Fanuc KAREL source: kb00158.KL

-- PROVISIONAL review KL for V770-1; original PC SHA256 021ea5336edb3704079312b4fe612844c061d565a7b6fe62d518488be7aab753
-- Incomplete behavior may be omitted. Consult companion uncertainty JSON. Do not deploy.
PROGRAM KB00158
%NOLOCKGROUP
BEGIN
  -- UNRESOLVED_PC offsets 5-12; opcodes 9D,23
  -- UNRESOLVED_PC offsets 17-24; opcodes 9D,23
  -- UNRESOLVED_PC offsets 29-45; opcodes 27,22,22,31
  -- UNRESOLVED_PC offsets 50-54; opcodes 7F
END KB00158
